TYPE ST_ComplexStruct :
STRUCT
	stSimple		:ST_SimpleStruct;
	stInte			:ST_Integrated1;
	sVer			:STRING ;
END_STRUCT
END_TYPE

(* stored: Version 1.1.0.1, ProductVersion 3.1.4024.15
   DUT ST_ComplexStruct: Id {19dad5f6-a26a-492e-8a1c-9016de129beb} *)
